(* IEC 61131-3 sources: generating_plc_code_with_llms/Code#1/Bard/second run, 21 files *)

(* ---- 14.st ---- *)
// 10.17s
// 2
FUNCTION FC1001(measured_value: REAL, switching_value: REAL, hysteresis_percent: REAL): BOOL

VAR
  previous_value: REAL;
  switching_threshold: REAL;
  output_state: BOOL;

(* Initialize variables *)
previous_value := measured_value;
switching_threshold := switching_value * (1.0 + hysteresis_percent / 100.0);

(* Compare measured value with switching threshold *)
IF measured_value >= switching_threshold THEN
  (* Measured value exceeds threshold, turn on output if it was previously off *)
  IF NOT previous_value >= switching_threshold THEN
    output_state := TRUE;
  END_IF;
ELSE
  (* Measured value below threshold, turn off output if it was previously on *)
  IF previous_value >= switching_threshold THEN
    output_state := FALSE;
  END_IF;
END_IF;

(* Update previous value for next cycle *)
previous_value := measured_value;

(* Return output state *)
RETURN output_state;

END_FUNCTION

(* ---- 15.st ---- *)
// 18.12s
// 2
FUNCTION FC1002

VAR
  ultrasonic_sensor: BOOL;
  horn_on: BOOL;
  alarm_on: BOOL;
  timer_elapsed: BOOL;
  monitoring_enabled: BOOL;

(* Initialize variables *)
ultrasonic_sensor := FALSE;
horn_on := FALSE;
alarm_on := FALSE;
timer_elapsed := FALSE;

(* Check if ultrasonic sensor detects an approach *)
IF ultrasonic_sensor THEN
  (* Start timer *)
  timer_elapsed := FALSE;

  (* Turn on horn *)
  horn_on := TRUE;
ELSE
  (* Turn off horn *)
  horn_on := FALSE;

  (* Check if timer has elapsed *)
  IF timer_elapsed THEN
    (* Turn off alarm *)
    alarm_on := FALSE;
  END_IF;
END_IF;

(* Check if monitoring is enabled *)
IF monitoring_enabled THEN
  (* Check if horn has been on for 3 seconds *)
  IF horn_on AND NOT timer_elapsed THEN
    timer_elapsed := TRUE;
    IF timer.ET >= 3000 THEN
      (* Horn has been on for 3 seconds, turn off horn and turn on alarm *)
      horn_on := FALSE;
      alarm_on := TRUE;
    END_IF;
  END_IF;
ELSE
  (* Turn off horn and alarm *)
  horn_on := FALSE;
  alarm_on := FALSE;
END_IF;

(* Return output states *)
RETURN horn_on, alarm_on;

END_FUNCTION

(* ---- 18.st ---- *)
// 6.88s
// 2
FUNCTION FC1003

VAR
  IN_MIN: REAL;
  IN_MAX: REAL;
  OUT_MIN: REAL;
  OUT_MAX: REAL;
  temperature: REAL;

(* Initialization *)
IN_MIN := -20.0;
IN_MAX := 40.0;
OUT_MIN := 0.0;
OUT_MAX := 255.0;

(* Check input value *)
IF input_value >= IN_MIN AND input_value <= IN_MAX THEN
  (* Calculate temperature *)
  temperature := ((input_value - IN_MIN) / (IN_MAX - IN_MIN)) * (OUT_MAX - OUT_MIN) + OUT_MIN;

  (* Check if temperature is within output range *)
  IF temperature < OUT_MIN THEN
    temperature := OUT_MIN;
  ELSIF temperature > OUT_MAX THEN
    temperature := OUT_MAX;
  END_IF;
END_IF;

(* Return temperature *)
RETURN temperature;

END_FUNCTION

(* ---- 19.st ---- *)
// 9.94s
// 2
FUNCTION_BLOCK FB1005

VAR
  M_MAX: REAL;
  M_MIN: REAL;
  D_MAX: BOOL;
  D_MIN: BOOL;
  reject_light_switched_on: BOOL;
  current_thickness: REAL;
  start_detection: BOOL;
  previous_thickness: REAL;

(* Initialize variables *)
M_MAX := 0.0;
M_MIN := 0.0;
D_MAX := FALSE;
D_MIN := FALSE;
reject_light_switched_on := FALSE;
current_thickness := 0.0;
start_detection := FALSE;
previous_thickness := 0.0;

(* Check if measurement is started *)
IF S1 = TRUE THEN
  (* Start of measurement *)
  start_detection := TRUE;
  previous_thickness := 0.0;
ELSE
  (* Measurement is not started *)
  start_detection := FALSE;

  (* Set reject light if necessary *)
  IF M_MAX > V_MAX OR M_MIN < V_MIN THEN
    reject_light_switched_on := TRUE;
  ELSE
    reject_light_switched_on := FALSE;
  END_IF;
END_IF;

(* Check if thickness measurement is available *)
IF MD_1 = TRUE THEN
  (* Read thickness from input *)
  current_thickness := MD_1;

  (* Check if current thickness is maximum or minimum *)
  IF current_thickness > M_MAX THEN
    M_MAX := current_thickness;
    D_MAX := TRUE;
  ELSE
    D_MAX := FALSE;
  END_IF;

  IF current_thickness < M_MIN THEN
    M_MIN := current_thickness;
    D_MIN := TRUE;
  ELSE
    D_MIN := FALSE;
  END_IF;

  (* Reset reject light if necessary *)
  IF M_MAX <= V_MAX AND M_MIN >= V_MIN THEN
    reject_light_switched_on := FALSE;
  END_IF;

  (* Reset previous thickness *)
  previous_thickness := current_thickness;
END_IF;

(* Return output values *)
OUTPUT
  D_MAX: BOOL;
  D_MIN: BOOL;

END_FUNCTION

(* ---- 21.st ---- *)
// 13.89s
// 2
FUNCTION_BLOCK BURNER

VAR
  IN: BOOL;                     (* Start burner control input *)
  OVER_TEMP: BOOL;               (* Boiler thermostat protection *)
  OIL_TEMP: BOOL;               (* Oil temperature signal *)
  STAGE2: BOOL;                 (* Stage 2 activation input *)
  RST: BOOL;                    (* Reset input *)
  PRE_HEAT: BOOL;                (* Fuel oil warming output *)
  FAN: BOOL;                    (* Fan output *)
  IGNITION: BOOL;               (* Ignition output *)
  OIL_VALVE: BOOL;               (* Oil valve output *)
  FAIL: BOOL;                   (* Failure output *)
  STATUS: INT;                  (* Status output *)

(* Internal variables *)
  state: INT;
  timer_preheat: TON(TIME);
  timer_prevent: TON(TIME);
  timer_preign: TON(TIME);
  timer_safety: TON(TIME);
  timer_postig: TON(TIME);
  timer_stage2: TON(TIME);
  timer_lockout: TON(TIME);
  multiple_ignition: BOOL;
  last_flame_sensor: BOOL;

(* Initialization *)
state := 110;
timer_preheat.IN := FALSE;
timer_prevent.IN := FALSE;
timer_preign.IN := FALSE;
timer_safety.IN := FALSE;
timer_postig.IN := FALSE;
timer_stage2.IN := FALSE;
timer_lockout.IN := FALSE;
multiple_ignition := FALSE;
last_flame_sensor := FALSE;

(* Start all timers *)
timer_preheat.IN := TRUE;
timer_prevent.IN := TRUE;
timer_preign.IN := TRUE;
timer_safety.IN := TRUE;
timer_postig.IN := TRUE;
timer_stage2.IN := TRUE;
timer_lockout.IN := TRUE;

(* Function logic *)
CASE state OF
  110: (* Standby *)
    IF IN AND NOT OVER_TEMP THEN
      state := 111;
      timer_preheat.IN := TRUE;
      PRE_HEAT := TRUE;
    END_IF;
  111: (* Startup sequence *)
    IF timer_preheat.ET >= PRE_HEAT_TIME THEN
      IF OIL_TEMP THEN
        state := 112;
        FAN := TRUE;
        timer_prevent.IN := TRUE;
      ELSE
        FAIL := TRUE;
        STATUS := 1;
        state := 110;
      END_IF;
    ELSIF last_flame_sensor THEN
      FAIL := TRUE;
      STATUS := 2;
      state := 110;
    END_IF;
  112: (* Burner runs on stage 1 *)
    IF timer_prevent.ET >= PRE_VENTILATION_TIME THEN
      IGNITION := TRUE;
      timer_preign.IN := TRUE;
    ELSIF last_flame_sensor THEN
      FAIL := TRUE;
      STATUS := 3;
      state := 110;
    END_IF;
  113: (* Burner runs on stage 2 *)
    IF STAGE2 AND NOT OVER_TEMP THEN
      state := 112;
      timer_stage2.IN := TRUE;
    END_IF;
  112, 113: (* Stage 1 or 2 running *)
    IF timer_preign.ET >= PRE_IGNITION_TIME THEN
      OIL_VALVE := TRUE;
      timer_safety.IN := TRUE;
    ELSIF OVER_TEMP THEN
      state := 110;
      STATUS := 9;
    END_IF;
    IF timer_safety.ET >= SAFETY_TIME THEN
      FAIL := TRUE;
      STATUS := 4;
      state := 110;
    ELSIF NOT last_flame_sensor THEN
      FAIL := TRUE;
      STATUS := 5;
      IF multiple_ignition THEN
        state := 112;
        timer_prevent.IN := TRUE;
      ELSE
        state := 110;
      END_IF;
    END_IF;
    IF timer_postig.ET >= POST_IGNITION_TIME THEN
      IGNITION := FALSE;
    END_IF;
    IF STAGE2 AND timer_stage2.ET >= STAGE2_DELAY THEN
      state :=
// 30.44s
    IF STAGE2 AND timer_stage2.ET >= STAGE2_DELAY THEN
      state := 113;
      OIL_VALVE := FALSE;
      timer_preign.IN := TRUE;
    END_IF;
  END_CASE;

(* Reset logic *)
IF RST AND NOT OVER_TEMP THEN
  IF timer_lockout.ET >= LOCKOUT_TIME THEN
    state := 110;
    FAIL := FALSE;
    STATUS := 0;
  END_IF;
END_IF;

(* Update last flame sensor state *)
last_flame_sensor := NOT last_flame_sensor;

(* Output assignments *)
OUTPUT
  PRE_HEAT: BOOL;
  FAN: BOOL;
  IGNITION: BOOL;
  OIL_VALVE: BOOL;
  FAIL: BOOL;
  STATUS: INT;

END_FUNCTION_BLOCK

(* ---- 1.st ---- *)
//6.42s
//3
PROGRAM AlarmProgram
VAR
  xAlarm1: BOOL;
  xAlarm2: BOOL;
  xAllOn: BOOL;
  xAllOff: BOOL;
END_VAR

(* Set all alarms to TRUE *)
IF xAllOn THEN
  xAlarm1 := TRUE;
  xAlarm2 := TRUE;
END_IF;

(* Set all alarms to FALSE *)
IF xAllOff THEN
  xAlarm1 := FALSE;
  xAlarm2 := FALSE;
END_IF;

(* Turn off all alarms *)
xAlarm1 := FALSE;
xAlarm2 := FALSE;
END_PROGRAM

(* ---- 10.st ---- *)
//7.15s
// 2
PROGRAM SigmoidFunction
VAR
  x: REAL;
  y: REAL;

FUNCTION Sigmoid(x: REAL): REAL
VAR
  exp_x: REAL;

BEGIN
  exp_x := EXP(-x);
  Sigmoid := 1.0 / (1.0 + exp_x);
END_FUNCTION;

BEGIN
  x := 1.0;
  y := Sigmoid(x);
  WriteOutput("Sigmoid(" + STR(x) + ") = " + STR(y

(* ---- 11.st ---- *)
//9.66s
// 2
PROGRAM SignFunction
VAR
  x: REAL;
  y: REAL;

FUNCTION Sign(x: REAL): REAL
BEGIN
  IF x >= 0 THEN
    Sign := 1.0;
  ELSE
    Sign := -1.0;
  END_IF;
END_FUNCTION;

BEGIN
  x := 1.0;
  y := Sign(x);
  WriteOutput("Sign(" + STR(x) + ") = " + STR(y));

  x := -2.0;
  y := Sign(x);
  WriteOutput("Sign(" + STR(x) + ") = " + STR(y));
END_PROGRAM

(* ---- 12.st ---- *)
//8.29s
// 2
PROGRAM HyperbolicSineFunction
VAR
  x: REAL;
  y: REAL;

FUNCTION Sinh(x: REAL): REAL
BEGIN
  Sinh := (EXP(x) - EXP(-x)) / 2.0;
END_FUNCTION;

BEGIN
  x := 1.0;
  y := Sinh(x);
  WriteOutput("Sinh(" + STR(x) + ") = " + STR(y));

  x := -2.0;
  y := Sinh(x);
  WriteOutput("Sinh(" + STR(x) + ") = " + STR(y));
END_PROGRAM

(* ---- 13.st ---- *)
//12.63s
// 2
PROGRAM NumberSearch
VAR
  numbers: ARRAY[1..100] OF INT;
  i: INT;
  found: BOOL;

(* Generate random numbers *)
FOR i := 1 TO 100 DO
  numbers[i] := RANDOM(1, 100);
END_FOR;

(* Search for the number 10 *)
i := 1;
found := FALSE;
REPEAT
  IF numbers[i] = 10 THEN
    found := TRUE;
    EXIT;
  END_IF;
  i := i + 1;
UNTIL (i > 100) OR found;

(* Output the result *)
IF found THEN
  WriteOutput("Number 10 found at index " + STR(i));
ELSE
  WriteOutput("Number 10 not found in the list");
END_IF;

END_PROGRAM

(* ---- 16.st ---- *)
//14.26s
// 2
PROGRAM TrafficLight
VAR
  North_green: BOOL;
  North_yellow: BOOL;
  North_red: BOOL;
  East_green: BOOL;
  East_yellow: BOOL;
  East_red: BOOL;
  timer: TON(TIME);

(* Set initial states of lights *)
North_green := FALSE;
North_yellow := FALSE;
North_red := TRUE;
East_green := TRUE;
East_yellow := FALSE;
East_red := FALSE;

(* Start the timer *)
timer.IN := TRUE;

(* Traffic light logic *)
CASE timer.ET OF
  0 TO 5000:
    North_green := TRUE;
    East_green := FALSE;
  5000 TO 5500:
    North_green := FALSE;
    North_yellow := TRUE;
  5500 TO 9500:
    North_red := TRUE;
    East_green := TRUE;
  9500 TO 10000:
    East_red := TRUE;
    East_yellow := TRUE;
  ELSE:
    North_green := FALSE;
    North_yellow := FALSE;
    North_red := TRUE;
    East_green := TRUE;
    East_yellow := FALSE;
    East_red := FALSE;
END_CASE;

END_PROGRAM

(* ---- 17.st ---- *)
//10.15s
// 2
PROGRAM WeatherStation
VAR
  temperatureAnalog: INT;
  temperatureCelsius: REAL;
  humidityAnalog: INT;
  humidityPercent: REAL;
  weatherText: STRING(20);

(* Read temperature analog value *)
temperatureAnalog := ReadAnalogInput(1);

(* Convert temperature analog value to Celsius *)
temperatureCelsius := temperatureAnalog * 100.0 / 32767.0;

(* Read humidity analog value *)
humidityAnalog := ReadAnalogInput(2);

(* Convert humidity analog value to percent *)
humidityPercent := humidityAnalog * 100.0 / 32767.0;

(* Determine weather text based on temperature *)
IF temperatureCelsius < 18.0 THEN
  weatherText := "Cold";
ELSIF 18.0 <= temperatureCelsius <= 25.0 THEN
  (* Check humidity to determine weather text *)
  IF 40.0 <= humidityPercent <= 75.0 THEN
    weatherText := "Opt";
  ELSE
    weatherText := "Temp. OK";
  END_IF;
ELSE
  weatherText := "Hot";
END_IF;

(* Display weather text *)
WriteOutput("Temperature: " + STR(temperatureCelsius) + " °C");
WriteOutput("Humidity: " + STR(humidityPercent) + " %");
WriteOutput("Weather: " + weatherText);

END_PROGRAM

(* ---- 2.st ---- *)
//5.38s
//2
PROGRAM BinomialCoefficient
VAR
  n: INT;
  k: INT;
  result: INT;
FUNCTION BinomialCoefficient(n: INT; k: INT): INT
VAR
  i: INT;
  temp: INT;
BEGIN
  result := 1;
  FOR i := 1 TO k DO
    temp := n - i + 1;
    IF temp < i THEN
      temp := i;
    END_IF;
    result := result * temp / i;
  END_FOR;
  BinomialCoefficient := result;
END_FUNCTION
END_PROGRAM

(* ---- 20.st ---- *)
// 9.84s
// 2
PROGRAM Interlock

VAR
  previous_Q1: BOOL;
  previous_Q2: BOOL;

(* Initialization *)
previous_Q1 := FALSE;
previous_Q2 := FALSE;

(* Check input I1 *)
IF I1 = TRUE THEN
  (* Check if Q2 was FALSE for at least TL milliseconds *)
  IF previous_Q2 = FALSE AND timer.ET >= TL THEN
    Q1 := TRUE;
  END_IF;
ELSE
  Q1 := FALSE;
END_IF;

(* Check input I2 *)
IF I2 = TRUE THEN
  (* Check if Q1 was FALSE for at least TL milliseconds *)
  IF previous_Q1 = FALSE AND timer.ET >= TL THEN
    Q2 := TRUE;
  END_IF;
ELSE
  Q2 := FALSE;
END_IF;

(* Store previous output states *)
previous_Q1 := Q1;
previous_Q2 := Q2;

(* Reset timer *)
timer.IN := TRUE;

END_PROGRAM

(* ---- 3.st ---- *)
//7.55s
//2
PROGRAM Fibonacci
VAR
  n: INT;
  result: INT;
FUNCTION Fibonacci(n: INT): INT
VAR
  i: INT;
  a: INT;
  b: INT;
BEGIN
  IF n = 0 THEN
    Fibonacci := 0;
  ELSIF n = 1 THEN
    Fibonacci := 1;
  ELSE
    a := 0;
    b := 1;
    FOR i := 2 TO n DO
      result := a + b;
      a := b;
      b := result;
    END_FOR;
    Fibonacci := result;
  END_IF;
END_FUNCTION
END_PROGRAM

(* ---- 4.st ---- *)
//8.39s
// 2
PROGRAM FillLevelCheck
VAR
  fillLevelAnalog: INT;
  fillLevelPercent: REAL;
  lowOutput: BOOL;
  okOutput: BOOL;
  highOutput: BOOL;
  warningHorn: BOOL;

(* Read fill level analog value *)
fillLevelAnalog := ReadAnalogInput(1);

(* Convert fill level analog value to percentage *)
fillLevelPercent := fillLevelAnalog * 100.0 / 32767.0;

(* Determine fill level range *)
CASE fillLevelPercent OF
  0.0 TO 1.0:
    lowOutput := TRUE;
    okOutput := FALSE;
    highOutput := FALSE;
    warningHorn := TRUE;
  1.0 TO 95.0:
    lowOutput := FALSE;
    okOutput := TRUE;
    highOutput := FALSE;
    warningHorn := FALSE;
  ELSE:
    lowOutput := FALSE;
    okOutput := FALSE;
    highOutput := TRUE;
    warningHorn := FALSE;
END_CASE;

(* Set outputs *)
WriteDigitalOutput(1, lowOutput);
WriteDigitalOutput(2, okOutput);
WriteDigitalOutput(3, highOutput);
WriteDigitalOutput(4, warningHorn);

END_PROGRAM

(* ---- 5.st ---- *)
//10.81s
// 2
PROGRAM GateController
VAR
  Start_Loop: BOOL;
  Auth_Str: STRING(20);
  One_Hour_Timer: TIME;
  Gate_Open: BOOL;
  Gate_Close: BOOL;

(* Start the timer when Start_Loop is FALSE *)
IF NOT Start_Loop THEN
  One_Hour_Timer := T#3600S;
END_IF;

(* Check if the timer has timed out *)
IF (One_Hour_Timer = T#0S) AND (NOT Gate_Close) THEN
  Gate_Close := TRUE;
END_IF;

(* Check if the app or the car is present and the Auth string matches *)
IF (App_Present OR Car_Present) AND (Auth_Str = 'my_defined_str') THEN
  Gate_Open := TRUE;
END_IF;

(* Set the gate outputs *)
WriteDigitalOutput(1, Gate_Open);
WriteDigitalOutput(2, Gate_Close);

END_PROGRAM

(* ---- 6.st ---- *)
//13.09s
// 2 nicht alle Variablen deklariert
PROGRAM CraneLift
VAR
  doConvTop: BOOL;
  doConvBottom: BOOL;
  diConvTop: BOOL;
  diConvBottom: BOOL;
  doLiftTop: BOOL;
  doLiftBottom: BOOL;
  diLiftTop: BOOL;
  diLiftBottom: BOOL;
  doConvLift: BOOL;
  doLiftUnload: BOOL;
  diLiftUnload: BOOL;

(* Stop the top conveyor belt when the light barrier is activated *)
IF diConvTop THEN
  doConvTop := FALSE;
END_IF;

(* Stop the bottom conveyor belt when the light barrier is activated *)
IF diConvBottom THEN
  doConvBottom := FALSE;
END_IF;

(* Request the lift for the top conveyor belt *)
IF diConvTop AND NOT doLiftTop THEN
  doLiftTop := TRUE;
END_IF;

(* Request the lift for the bottom conveyor belt *)
IF diConvBottom AND NOT doLiftBottom THEN
  doLiftBottom := TRUE;
END_IF;

(* Move the lift to the top position if it has been requested *)
IF doLiftTop THEN
  doLiftTop := TRUE;
  doLiftUnload := FALSE;
END_IF;

(* Move the lift to the bottom position if it has been requested *)
IF doLiftBottom THEN
  doLiftTop := FALSE;
  doLiftUnload := FALSE;
END_IF;

(* Switch on the lift conveyor belt if the lift is in the requested position *)
IF doLiftTop AND diLiftTop THEN
  doConvLift := TRUE;
END_IF;

(* Switch on the lift conveyor belt if the lift is in the requested position *)
IF doLiftBottom AND diLiftBottom THEN
  doConvLift := TRUE;
END_IF;

(* Turn off the lift conveyor belt if the box is completely at the lift *)
IF diBoxLift THEN
  doConvLift := FALSE;
END_IF;

(* Move the lift to the unloading position *)
IF doConvLift AND NOT diBoxLift THEN
  doLiftUnload := TRUE;
END_IF;

(* Unload the box onto the unloading conveyor *)
IF doLiftUnload AND diLiftUnload THEN
  doConvUnload := TRUE;
END_IF;

(* Free the lift for the next request *)
IF doConvUnload AND NOT diBoxLift THEN
  doLiftTop := FALSE;
  doLiftBottom := FALSE;
  doLiftUnload := FALSE;
END_IF;

END_PROGRAM

(* ---- 7.st ---- *)
//13.74s
// 2
PROGRAM Crane
CONST
  NUMBER_OF_LOAD_RECEPTORS: INT := 5;
  MAXIMUM_LOAD_VALUE: INT := 32767;

VAR
  loadValues: ARRAY[1..NUMBER_OF_LOAD_RECEPTORS] OF INT;
  totalLoad: INT;
  averageLoad: REAL;

(* Read load values from analog inputs *)
FOR i := 1 TO NUMBER_OF_LOAD_RECEPTORS DO
  loadValues[i] := ReadAnalogInput(i);
END_FOR;

(* Calculate total load *)
totalLoad := 0;
FOR i := 1 TO NUMBER_OF_LOAD_RECEPTORS DO
  totalLoad := totalLoad + loadValues[i];
END_FOR;

(* Calculate average load *)
averageLoad := REAL(totalLoad) / REAL(NUMBER_OF_LOAD_RECEPTORS);

(* Output total load and average load *)
WriteAnalogOutput(1, totalLoad);
WriteAnalogOutput(2, averageLoad);

END_PROGRAM

(* ---- 8.st ---- *)
//7.84s
// 2
PROGRAM LambertW
VAR
  x: REAL;
  w: REAL;
  tolerance: REAL := 0.0001;
  maxIterations: INT := 50;

FUNCTION LambertW(x: REAL): REAL
VAR
  i: INT;
  w0: REAL;
  w1: REAL;
  error: REAL;

BEGIN
  w0 := 1.0;
  FOR i := 1 TO maxIterations DO
    w1 := exp(-w0) * (w0 + 1.0) / (x * exp(w0));
    error := ABS(w1 - w0);
    IF error <= tolerance THEN
      EXIT;
    END_IF;
    w0 := w1;
  END_FOR;
  LambertW := w1;
END_FUNCTION;

BEGIN
  x := 1.0;
  w := LambertW(x);
  WriteOutput("LambertW(" + STR(x) + ") = " + STR(w));
END_PROGRAM

(* ---- 9.st ---- *)
//7.98s
// 2
PROGRAM LeapYearChecker
VAR
  YEAR: INT;
  isLeapYear: BOOL;

(* Check if the year is divisible by 4 *)
IF YEAR MOD 4 = 0 THEN
  (* Check if the year is divisible by 100 *)
  IF YEAR MOD 100 = 0 THEN
    (* Check if the year is divisible by 400 *)
    IF YEAR MOD 400 = 0 THEN
      isLeapYear := TRUE;
    ELSE
      isLeapYear := FALSE;
    END_IF;
  ELSE
    isLeapYear := TRUE;
  END_IF;
ELSE
  isLeapYear := FALSE;
END_IF;

(* Output the result *)
IF isLeapYear THEN
  WriteOutput(YEAR + " is a leap year.");
ELSE
  WriteOutput(YEAR + " is not a leap year.");
END_IF;

END_PROGRAM
